//{attribute 'qualified_only'}
VAR_GLOBAL
	bDraaipoortVolledigOpenDicht	AT %Q*	: BOOL;
	bDraaipoortVoetgangerOpenDicht	AT %Q*	: BOOL;
END_VAR

(* stored: Version 1.1.0.1
   GVL GVL_Draaipoort: Id {d05611e3-9ff0-43f1-81e5-cfa2a8daaf3e} *)
